TYPE "udt_Rollformer_Pers"
VERSION : 0.1
// Block: udt_Rollformer_Pers
   STRUCT
      Machine : Struct
         Par : Struct
            ExtraLow_Enable : Bool;
            ExtraLow_VelPercentage : Real;
         END_STRUCT;
      END_STRUCT;
      Feed : Struct
         Par : PositioningMachine_Par;
         Pers_Data : PositioningMachine_DataPers;
      END_STRUCT;
   END_STRUCT;

END_TYPE
